TYPE ST_GCSpinAxisMoveAbsStatus EXTENDS ST_ServiceStatusBase :
STRUCT
END_STRUCT
END_TYPE

(* stored: Version 1.1.0.1, ProductVersion 3.1.4026.18
   DUT ST_GCSpinAxisMoveAbsStatus: Id {c8f84dfe-7f7b-4980-b837-341c09bf5471} *)
